// TIA Portal V20 export
TYPE "LKinCtrl_typeConfiguration"
   STRUCT
      offsetParameter : Array[1.."LKINCTRL_NO_OF_OFFSETS"] of "LKinCtrl_typeContourOffsetParameter";   // offset parameter settings
      conveyorParameter : Array[1.."LKINCTRL_NO_OF_CONVEYOR"] of "LKinCtrl_typeConveyorConfiguration";   // conveyor parameter settings
      userFrames : Array["LKINCTRL_CS_NO_OF_FIRST_USER_FRAME".."LKINCTRL_CS_NO_OF_LAST_USER_FRAME"] of "LKinCtrl_typeFrame";   // user frames configuration
      workspaceZones : Array[1.."LKINCTRL_NO_OF_ZONES"] of "LKinCtrl_typeWorkspaceZoneDefinition";   // workspace zone configurations
      kinematicsZones : Array[1.."LKINCTRL_NO_OF_ZONES"] of "LKinCtrl_typeKinematicsZoneDefinition";   // kinematics zone configuration
      stopMode : DInt;   // MC_GroupStop dynamics; 0: stop with dynamics of active motion job; 1: stop with maximum kinematics dynamics (dynamics adaption still effective); 10: stop with dynamics of active motion job and desync conveyor; 11: stop with maximum kinematics dynamics and desync conveyor
      interruptMode : DInt;   // MC_GroupInterrupt dynamics; 0: interrupt with dynamics of active motion job; 1: interrupt with maximum kinematics dynamics (dynamics adaption still effective)
   END_STRUCT;
END_TYPE
